KUKA KRL data list: vw_user.dat

&ACCESS RV
&PARAM TPVW_VERSION = 3.3.5
DEFDAT  VW_USER
ENDDAT
